FUNCTION_BLOCK FB_TestCase03Station EXTENDS FB_TestCaseBase
VAR
	fbTestStation	: FB_TestStation;
	stTestStationIO : ST_TestStation_IO;
	eStState		: E_ComponentState;
	iTest			: INT;
	bInit			: BOOL;
	bEnable			: BOOL := TRUE;
	bSafetyOk		: BOOL := TRUE;
	bTestOk 		: BOOL := FALSE;
END_VAR

{attribute 'object_name' := 'Run'}
METHOD Run : E_TestCaseState
// init state in base
Run := SUPER^.Run();
IF Run <> E_TestCaseState.eTestCaseState_running THEN
	RETURN;
END_IF

// test
fbTestStation.Enable := bEnable;
fbTestStation.SafetyOk := bSafetyOk;
fbTestStation();
CASE iTest OF
	0:	// init / idle / no Test
		IF NOT bInit THEN
			iTest := 1;
			RETURN;
		END_IF
		
	10:	// init Station
		bInit := TRUE;
		fbTestStation.stIO := stTestStationIO;		
		
	20:	// reset
		fbTestStation.Reset();
		
	30:	// execute command
		;//stRes := fbTestStation.ExecuteCmd(stCmd);
		
END_CASE
iTest := 0;

// update result and state
IF bTestOk THEN
	eResult := E_TestResult.eTestResult_ok; //check log files!
	eState := E_TestCaseState.eTestCaseState_finished;
END_IF

Run := eState;
END_METHOD

END_FUNCTION_BLOCK

(* stored: Version 1.1.0.1, ProductVersion 3.1.4024.4
   POU FB_TestCase03Station: Id {fa6cfa2c-c98a-45a5-bcff-7d1185d8276d}, SpecialFunc None
   Method Run: Id {ea34b146-6ad7-44d8-a6ee-17fd74278a52} *)
